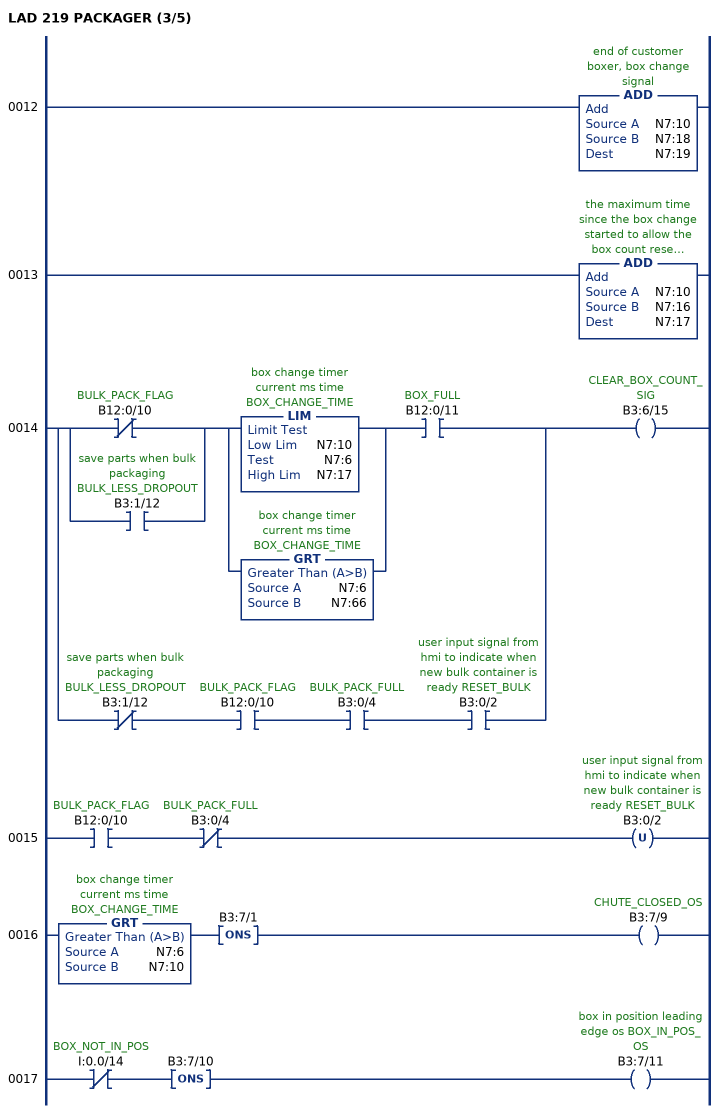
% Rung: 12 %
SOR ADD N7:10 N7:18 N7:19 EOR
%   N7:10  CHUTE_CLOSED_TIME  "time at which chute door is considered closed" %
%   N7:18  CHANGE_BOX_SIG_TIME  "customer boxer change box signal time" %
%   N7:19  "end of customer boxer, box change signal" %
% Rung: 13 %
SOR ADD N7:10 N7:16 N7:17 EOR
%   N7:10  CHUTE_CLOSED_TIME  "time at which chute door is considered closed" %
%   N7:16  RESET_COUNT_SIG_TIME  "maximum length of time to hold box count reset signal on" %
%   N7:17  "the maximum time since the box change started to allow the box count reset signal" %
% Rung: 14 %
SOR BST BST XIO B12:0/10 NXB XIC B3:1/12 BND BST LIM N7:10 N7:6 N7:17 NXB GRT N7:6 N7:66 BND XIC B12:0/11 NXB XIO B3:1/12 XIC B12:0/10 XIC B3:0/4 XIC B3:0/2 BND OTE B3:6/15 EOR
%   B12:0/10  BULK_PACK_FLAG %
%   B3:1/12  BULK_LESS_DROPOUT  "save parts when bulk packaging" %
%   N7:10  CHUTE_CLOSED_TIME  "time at which chute door is considered closed" %
%   N7:6  BOX_CHANGE_TIME  "box change timer current ms time" %
%   N7:17  "the maximum time since the box change started to allow the box count reset signal" %
%   B12:0/11  BOX_FULL %
%   B3:0/4  BULK_PACK_FULL %
%   B3:0/2  RESET_BULK  "user input signal from hmi to indicate when new bulk container is ready" %
%   B3:6/15  CLEAR_BOX_COUNT_SIG %
% Rung: 15 %
SOR XIC B12:0/10 XIO B3:0/4 OTU B3:0/2 EOR
%   B12:0/10  BULK_PACK_FLAG %
%   B3:0/4  BULK_PACK_FULL %
%   B3:0/2  RESET_BULK  "user input signal from hmi to indicate when new bulk container is ready" %
% Rung: 16 %
SOR GRT N7:6 N7:10 ONS B3:7/1 OTE B3:7/9 EOR
%   N7:6  BOX_CHANGE_TIME  "box change timer current ms time" %
%   N7:10  CHUTE_CLOSED_TIME  "time at which chute door is considered closed" %
%   B3:7/9  CHUTE_CLOSED_OS %
% Rung: 17 %
SOR XIO I:0.0/14 ONS B3:7/10 OTE B3:7/11 EOR
%   I:0.0/14  BOX_NOT_IN_POS %
%   B3:7/11  BOX_IN_POS_OS  "box in position leading edge os" %

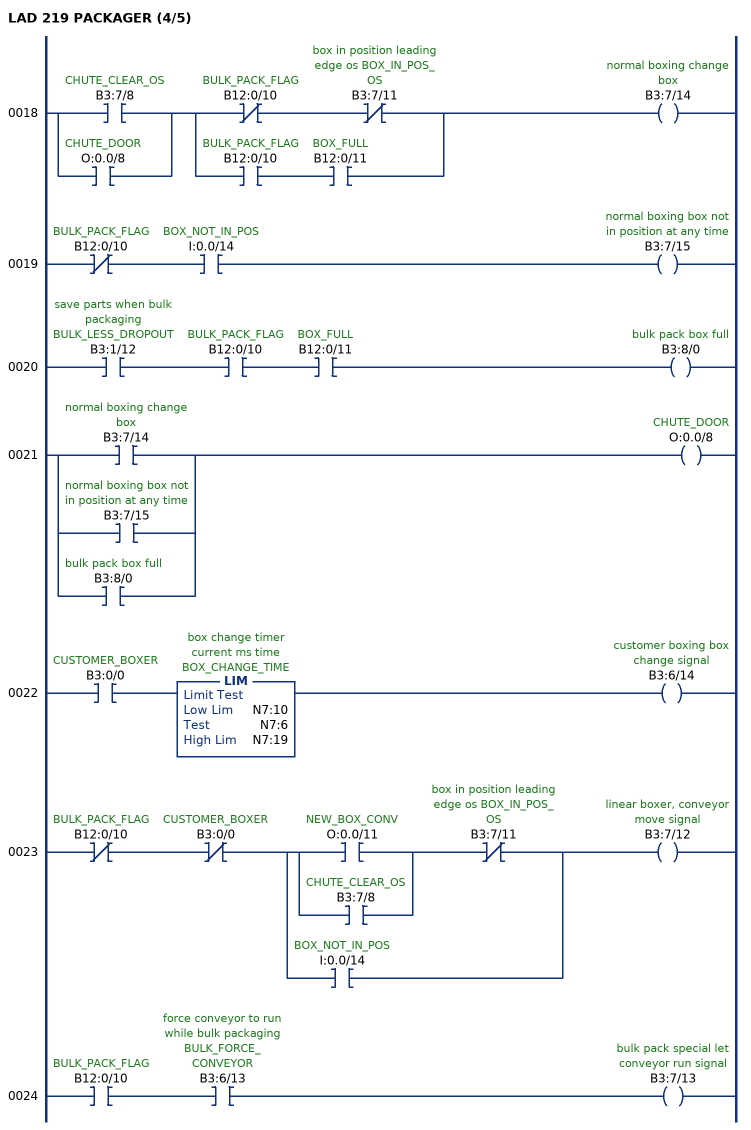
% Rung: 18 %
SOR BST XIC B3:7/8 NXB XIC O:0.0/8 BND BST XIO B12:0/10 XIO B3:7/11 NXB XIC B12:0/10 XIC B12:0/11 BND OTE B3:7/14 EOR
%   B3:7/8  CHUTE_CLEAR_OS %
%   O:0.0/8  CHUTE_DOOR %
%   B12:0/10  BULK_PACK_FLAG %
%   B3:7/11  BOX_IN_POS_OS  "box in position leading edge os" %
%   B12:0/11  BOX_FULL %
%   B3:7/14  "normal boxing change box" %
% Rung: 19 %
SOR XIO B12:0/10 XIC I:0.0/14 OTE B3:7/15 EOR
%   B12:0/10  BULK_PACK_FLAG %
%   I:0.0/14  BOX_NOT_IN_POS %
%   B3:7/15  "normal boxing box not in position at any time" %
% Rung: 20 %
SOR XIC B3:1/12 XIC B12:0/10 XIC B12:0/11 OTE B3:8/0 EOR
%   B3:1/12  BULK_LESS_DROPOUT  "save parts when bulk packaging" %
%   B12:0/10  BULK_PACK_FLAG %
%   B12:0/11  BOX_FULL %
%   B3:8/0  "bulk pack box full" %
% Rung: 21 %
SOR BST XIC B3:7/14 NXB XIC B3:7/15 NXB XIC B3:8/0 BND OTE O:0.0/8 EOR
%   B3:7/14  "normal boxing change box" %
%   B3:7/15  "normal boxing box not in position at any time" %
%   B3:8/0  "bulk pack box full" %
%   O:0.0/8  CHUTE_DOOR %
% Rung: 22 %
SOR XIC B3:0/0 LIM N7:10 N7:6 N7:19 OTE B3:6/14 EOR
%   B3:0/0  CUSTOMER_BOXER %
%   N7:10  CHUTE_CLOSED_TIME  "time at which chute door is considered closed" %
%   N7:6  BOX_CHANGE_TIME  "box change timer current ms time" %
%   N7:19  "end of customer boxer, box change signal" %
%   B3:6/14  "customer boxing box change signal" %
% Rung: 23 %
SOR XIO B12:0/10 XIO B3:0/0 BST BST XIC O:0.0/11 NXB XIC B3:7/8 BND XIO B3:7/11 NXB XIC I:0.0/14 BND OTE B3:7/12 EOR
%   B12:0/10  BULK_PACK_FLAG %
%   B3:0/0  CUSTOMER_BOXER %
%   O:0.0/11  NEW_BOX_CONV %
%   B3:7/8  CHUTE_CLEAR_OS %
%   B3:7/11  BOX_IN_POS_OS  "box in position leading edge os" %
%   I:0.0/14  BOX_NOT_IN_POS %
%   B3:7/12  "linear boxer, conveyor move signal" %
% Rung: 24 %
SOR XIC B12:0/10 XIC B3:6/13 OTE B3:7/13 EOR
%   B12:0/10  BULK_PACK_FLAG %
%   B3:6/13  BULK_FORCE_CONVEYOR  "force conveyor to run while bulk packaging" %
%   B3:7/13  "bulk pack special let conveyor run signal" %

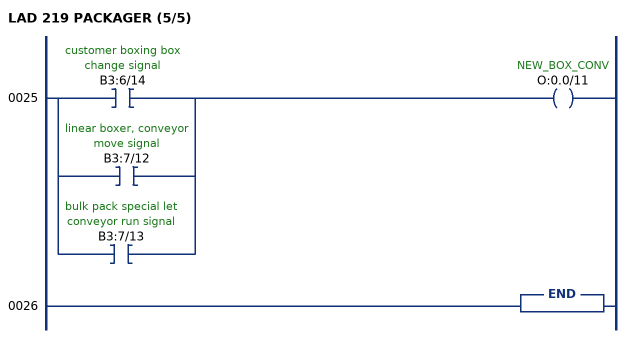
% Rung: 25 %
SOR BST XIC B3:6/14 NXB XIC B3:7/12 NXB XIC B3:7/13 BND OTE O:0.0/11 EOR
%   B3:6/14  "customer boxing box change signal" %
%   B3:7/12  "linear boxer, conveyor move signal" %
%   B3:7/13  "bulk pack special let conveyor run signal" %
%   O:0.0/11  NEW_BOX_CONV %
% Rung: 26 %
SOR END EOR

LADDER 220 "NO PACKAGE"
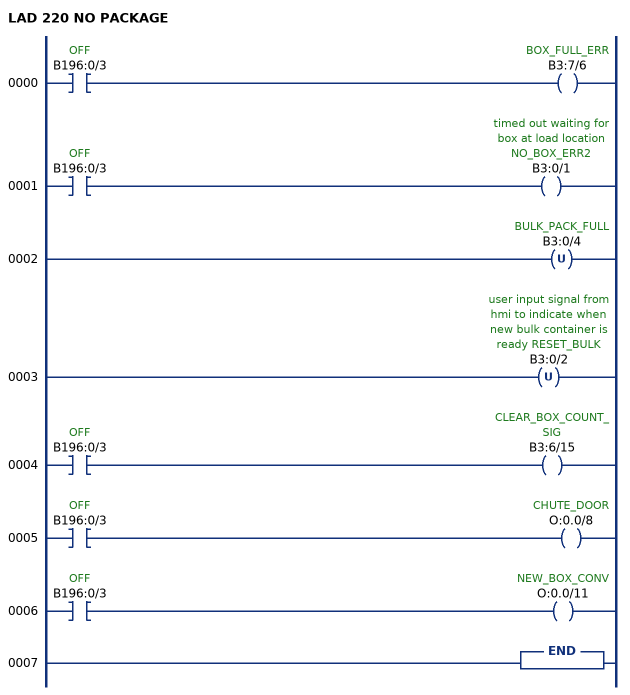
% Rung: 0 %
SOR XIC B196:0/3 OTE B3:7/6 EOR
%   B196:0/3  OFF %
%   B3:7/6  BOX_FULL_ERR %
% Rung: 1 %
SOR XIC B196:0/3 OTE B3:0/1 EOR
%   B196:0/3  OFF %
%   B3:0/1  NO_BOX_ERR2  "timed out waiting for box at load location" %
% Rung: 2 %
SOR OTU B3:0/4 EOR
%   B3:0/4  BULK_PACK_FULL %
% Rung: 3 %
SOR OTU B3:0/2 EOR
%   B3:0/2  RESET_BULK  "user input signal from hmi to indicate when new bulk container is ready" %
% Rung: 4 %
SOR XIC B196:0/3 OTE B3:6/15 EOR
%   B196:0/3  OFF %
%   B3:6/15  CLEAR_BOX_COUNT_SIG %
% Rung: 5 %
SOR XIC B196:0/3 OTE O:0.0/8 EOR
%   B196:0/3  OFF %
%   O:0.0/8  CHUTE_DOOR %
% Rung: 6 %
SOR XIC B196:0/3 OTE O:0.0/11 EOR
%   B196:0/3  OFF %
%   O:0.0/11  NEW_BOX_CONV %
% Rung: 7 %
SOR END EOR

LADDER 222 "RATE1"
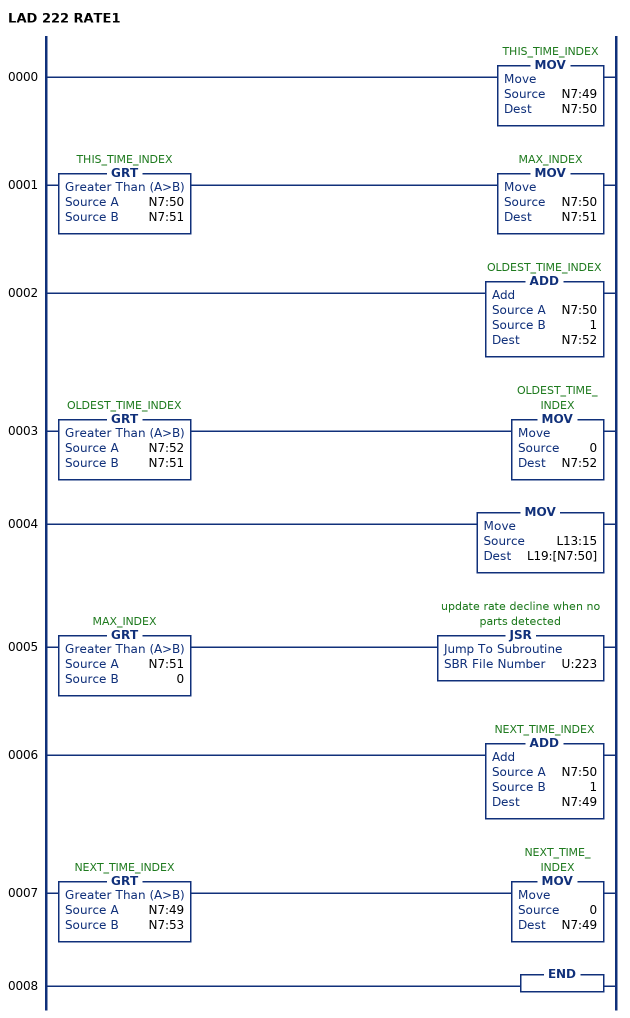
% Rung: 0 %
SOR MOV N7:49 N7:50 EOR
%   N7:49  NEXT_TIME_INDEX %
%   N7:50  THIS_TIME_INDEX %
% Rung: 1 %
SOR GRT N7:50 N7:51 MOV N7:50 N7:51 EOR
%   N7:50  THIS_TIME_INDEX %
%   N7:51  MAX_INDEX %
% Rung: 2 %
SOR ADD N7:50 1 N7:52 EOR
%   N7:50  THIS_TIME_INDEX %
%   N7:52  OLDEST_TIME_INDEX %
% Rung: 3 %
SOR GRT N7:52 N7:51 MOV 0 N7:52 EOR
%   N7:52  OLDEST_TIME_INDEX %
%   N7:51  MAX_INDEX %
% Rung: 4 %
SOR MOV L13:15 L19:[N7:50] EOR
%   L13:15  THE_TIME %
%   N7:50  THIS_TIME_INDEX %
% Rung: 5 %
SOR GRT N7:51 0 JSR U:223 EOR
%   N7:51  MAX_INDEX %
%   U:223  "update rate decline when no parts detected" %
% Rung: 6 %
SOR ADD N7:50 1 N7:49 EOR
%   N7:50  THIS_TIME_INDEX %
%   N7:49  NEXT_TIME_INDEX %
% Rung: 7 %
SOR GRT N7:49 N7:53 MOV 0 N7:49 EOR
%   N7:49  NEXT_TIME_INDEX %
%   N7:53  UPPER_INDEX_LIMIT %
% Rung: 8 %
SOR END EOR

LADDER 223 "RATE2"
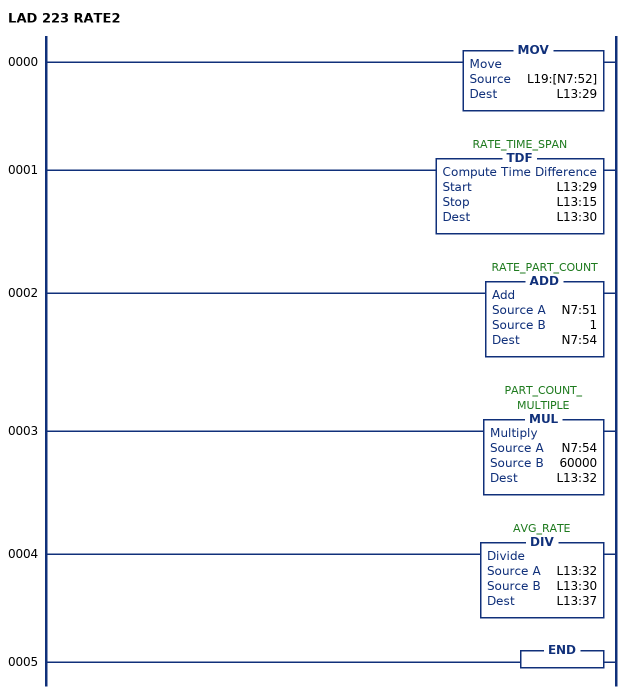
% Rung: 0 %
SOR MOV L19:[N7:52] L13:29 EOR
%   N7:52  OLDEST_TIME_INDEX %
% Rung: 1 %
SOR TDF L13:29 L13:15 L13:30 EOR
%   L13:15  THE_TIME %
%   L13:30  RATE_TIME_SPAN %
% Rung: 2 %
SOR ADD N7:51 1 N7:54 EOR
%   N7:51  MAX_INDEX %
%   N7:54  RATE_PART_COUNT %
% Rung: 3 %
SOR MUL N7:54 60000 L13:32 EOR
%   N7:54  RATE_PART_COUNT %
%   L13:32  PART_COUNT_MULTIPLE %
% Rung: 4 %
SOR DIV L13:32 L13:30 L13:37 EOR
%   L13:32  PART_COUNT_MULTIPLE %
%   L13:30  RATE_TIME_SPAN %
%   L13:37  AVG_RATE %
% Rung: 5 %
SOR END EOR

LADDER 224 "RESET RATE"
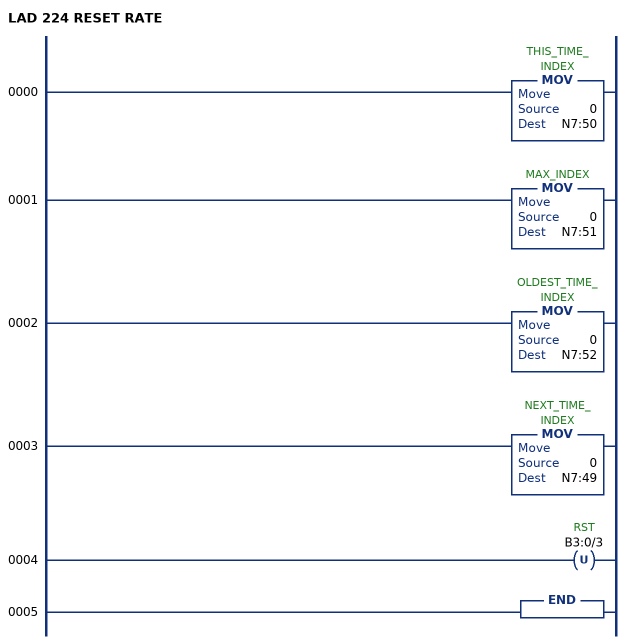
% Rung: 0 %
SOR MOV 0 N7:50 EOR
%   N7:50  THIS_TIME_INDEX %
% Rung: 1 %
SOR MOV 0 N7:51 EOR
%   N7:51  MAX_INDEX %
% Rung: 2 %
SOR MOV 0 N7:52 EOR
%   N7:52  OLDEST_TIME_INDEX %
% Rung: 3 %
SOR MOV 0 N7:49 EOR
%   N7:49  NEXT_TIME_INDEX %
% Rung: 4 %
SOR OTU B3:0/3 EOR
%   B3:0/3  RST %
% Rung: 5 %
SOR END EOR

LADDER 240 "NP STOP"
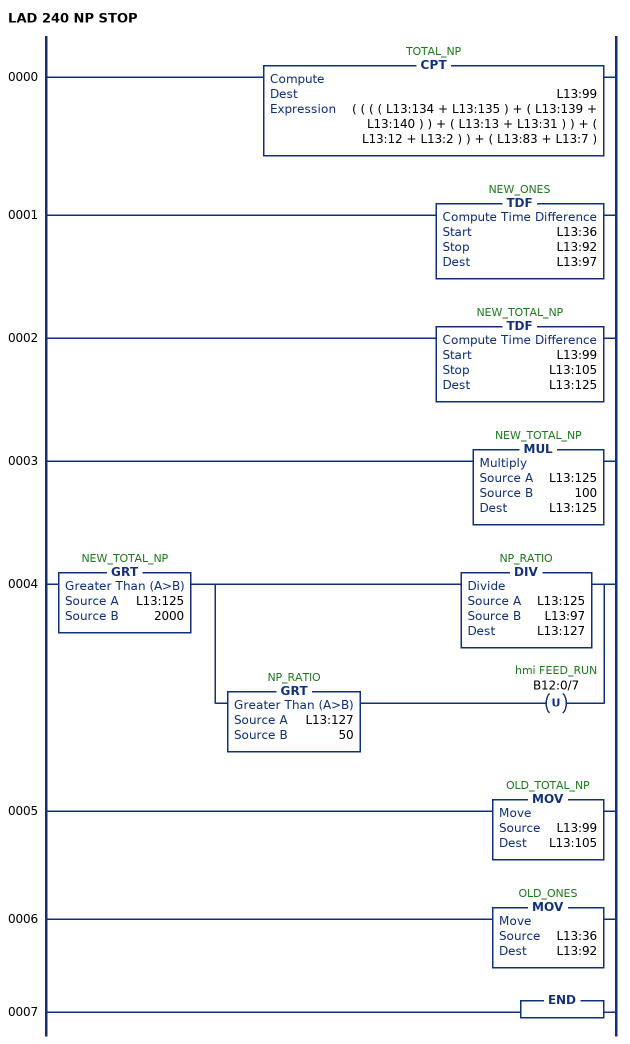
% Rung: 0 %
SOR CPT L13:99 " ( ( ( ( L13:134 + L13:135 ) + ( L13:139 + L13:140 ) ) + ( L13:13 + L13:31 ) ) + ( L13:12 + L13:2 ) ) + ( L13:83 + L13:7 ) " EOR
%   L13:99  TOTAL_NP %
%   L13:134  "too wide bottom" %
%   L13:135  "too close bottom" %
%   L13:139  "too close top count" %
%   L13:140  "too wide top count" %
%   L13:13  SKIP1  "skipped 1 count" %
%   L13:31  SKIP5  "skipped 5 count" %
%   L13:12  SKIP6  "skipped 6 count" %
%   L13:2  INS1_FAIL_COUNT %
%   L13:83  INS5_FAIL_COUNT %
%   L13:7  INS6_FAIL_COUNT %
% Rung: 1 %
SOR TDF L13:36 L13:92 L13:97 EOR
%   L13:36  ONES %
%   L13:92  OLD_ONES %
%   L13:97  NEW_ONES %
% Rung: 2 %
SOR TDF L13:99 L13:105 L13:125 EOR
%   L13:99  TOTAL_NP %
%   L13:105  OLD_TOTAL_NP %
%   L13:125  NEW_TOTAL_NP %
% Rung: 3 %
SOR MUL L13:125 100 L13:125 EOR
%   L13:125  NEW_TOTAL_NP %
% Rung: 4 %
SOR GRT L13:125 2000 BST DIV L13:125 L13:97 L13:127 NXB GRT L13:127 50 OTU B12:0/7 BND EOR
%   L13:125  NEW_TOTAL_NP %
%   L13:97  NEW_ONES %
%   L13:127  NP_RATIO %
%   B12:0/7  FEED_RUN  "hmi" %
% Rung: 5 %
SOR MOV L13:99 L13:105 EOR
%   L13:99  TOTAL_NP %
%   L13:105  OLD_TOTAL_NP %
% Rung: 6 %
SOR MOV L13:36 L13:92 EOR
%   L13:36  ONES %
%   L13:92  OLD_ONES %
% Rung: 7 %
SOR END EOR

LADDER 246 "SPEED BOT"    % high speed %
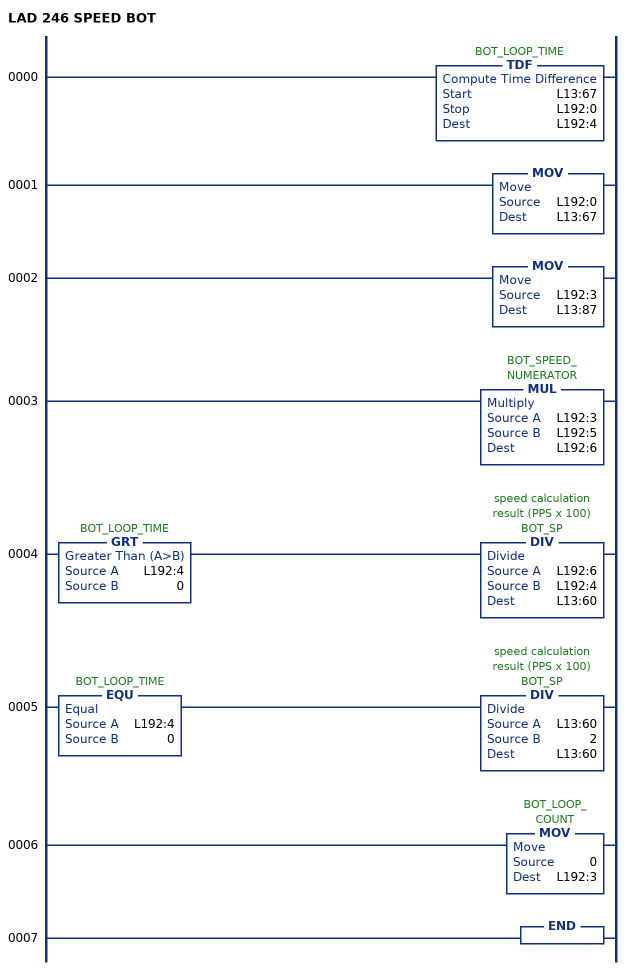
% Rung: 0 %
SOR TDF L13:67 L192:0 L192:4 EOR
%   L192:0  BOT_THIS_TIME  "rtc bot belt movement event time" %
%   L192:4  BOT_LOOP_TIME %
% Rung: 1 %
SOR MOV L192:0 L13:67 EOR
%   L192:0  BOT_THIS_TIME  "rtc bot belt movement event time" %
% Rung: 2 %
SOR MOV L192:3 L13:87 EOR
%   L192:3  BOT_LOOP_COUNT %
% Rung: 3 %
SOR MUL L192:3 L192:5 L192:6 EOR
%   L192:3  BOT_LOOP_COUNT %
%   L192:5  TKS_PER_SECOND %
%   L192:6  BOT_SPEED_NUMERATOR %
% Rung: 4 %
SOR GRT L192:4 0 DIV L192:6 L192:4 L13:60 EOR
%   L192:4  BOT_LOOP_TIME %
%   L192:6  BOT_SPEED_NUMERATOR %
%   L13:60  BOT_SP  "speed calculation result (PPS x 100)" %
% Rung: 5 %
SOR EQU L192:4 0 DIV L13:60 2 L13:60 EOR
%   L192:4  BOT_LOOP_TIME %
%   L13:60  BOT_SP  "speed calculation result (PPS x 100)" %
% Rung: 6 %
SOR MOV 0 L192:3 EOR
%   L192:3  BOT_LOOP_COUNT %
% Rung: 7 %
SOR END EOR

LADDER 248 "SPEED TOP"    % high speed %
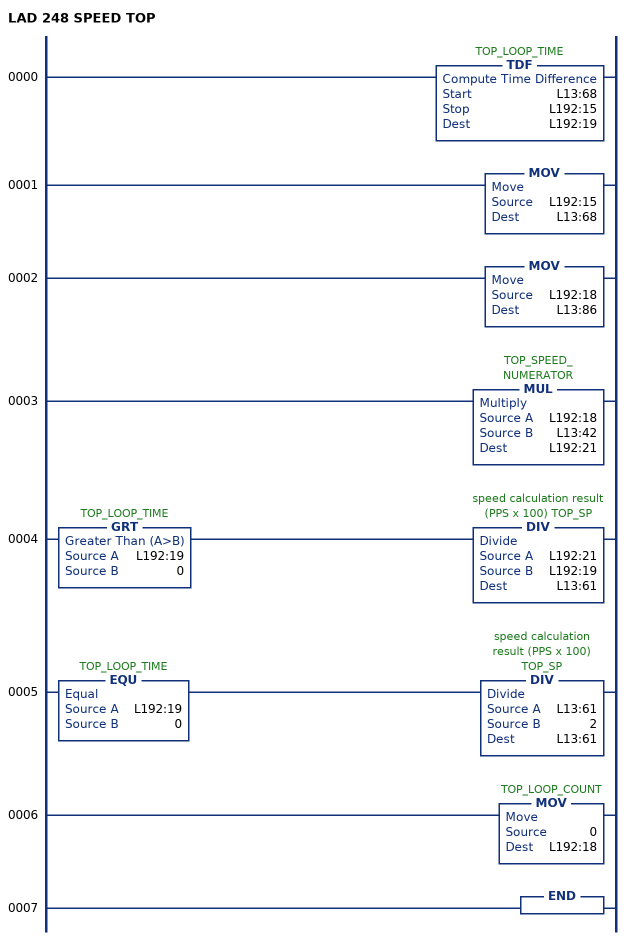
% Rung: 0 %
SOR TDF L13:68 L192:15 L192:19 EOR
%   L192:15  TOP_THIS_TIME  "rtc top belt movement event time" %
%   L192:19  TOP_LOOP_TIME %
% Rung: 1 %
SOR MOV L192:15 L13:68 EOR
%   L192:15  TOP_THIS_TIME  "rtc top belt movement event time" %
% Rung: 2 %
SOR MOV L192:18 L13:86 EOR
%   L192:18  TOP_LOOP_COUNT %
% Rung: 3 %
SOR MUL L192:18 L13:42 L192:21 EOR
%   L192:18  TOP_LOOP_COUNT %
%   L192:21  TOP_SPEED_NUMERATOR %
% Rung: 4 %
SOR GRT L192:19 0 DIV L192:21 L192:19 L13:61 EOR
%   L192:19  TOP_LOOP_TIME %
%   L192:21  TOP_SPEED_NUMERATOR %
%   L13:61  TOP_SP  "speed calculation result (PPS x 100)" %
% Rung: 5 %
SOR EQU L192:19 0 DIV L13:61 2 L13:61 EOR
%   L192:19  TOP_LOOP_TIME %
%   L13:61  TOP_SP  "speed calculation result (PPS x 100)" %
% Rung: 6 %
SOR MOV 0 L192:18 EOR
%   L192:18  TOP_LOOP_COUNT %
% Rung: 7 %
SOR END EOR

LADDER 250 "P BOT"    % high speed %
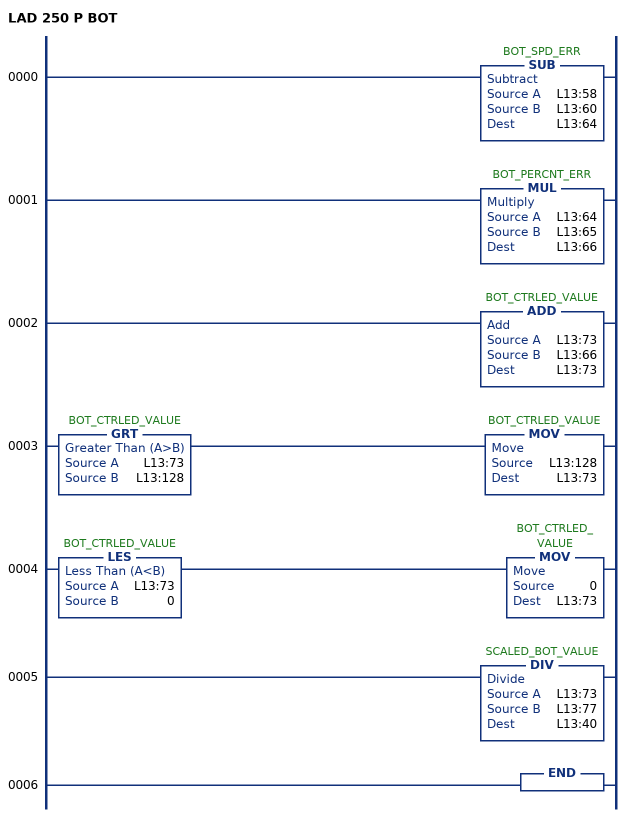
% Rung: 0 %
SOR SUB L13:58 L13:60 L13:64 EOR
%   L13:58  BOT_SPD_SETPOINT %
%   L13:60  BOT_SP  "speed calculation result (PPS x 100)" %
%   L13:64  BOT_SPD_ERR %
% Rung: 1 %
SOR MUL L13:64 L13:65 L13:66 EOR
%   L13:64  BOT_SPD_ERR %
%   L13:65  POS5SHIFT %
%   L13:66  BOT_PERCNT_ERR %
% Rung: 2 %
SOR ADD L13:73 L13:66 L13:73 EOR
%   L13:73  BOT_CTRLED_VALUE %
%   L13:66  BOT_PERCNT_ERR %
% Rung: 3 %
SOR GRT L13:73 L13:128 MOV L13:128 L13:73 EOR
%   L13:73  BOT_CTRLED_VALUE %
%   L13:128  "how much top has shifted since measurment" %
% Rung: 4 %
SOR LES L13:73 0 MOV 0 L13:73 EOR
%   L13:73  BOT_CTRLED_VALUE %
% Rung: 5 %
SOR DIV L13:73 L13:77 L13:40 EOR
%   L13:73  BOT_CTRLED_VALUE %
%   L13:40  SCALED_BOT_VALUE %
% Rung: 6 %
SOR END EOR

LADDER 252 "P TOP"    % high speed %
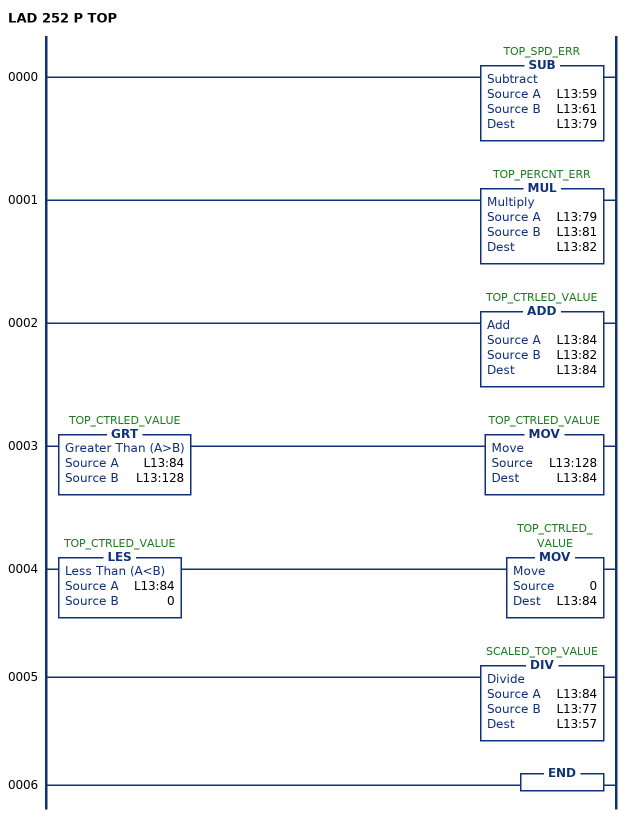
% Rung: 0 %
SOR SUB L13:59 L13:61 L13:79 EOR
%   L13:59  TOP_SPD_SETPOINT %
%   L13:61  TOP_SP  "speed calculation result (PPS x 100)" %
%   L13:79  TOP_SPD_ERR %
% Rung: 1 %
SOR MUL L13:79 L13:81 L13:82 EOR
%   L13:79  TOP_SPD_ERR %
%   L13:81  TOP_FDBK_RATIO %
%   L13:82  TOP_PERCNT_ERR %
% Rung: 2 %
SOR ADD L13:84 L13:82 L13:84 EOR
%   L13:84  TOP_CTRLED_VALUE %
%   L13:82  TOP_PERCNT_ERR %
% Rung: 3 %
SOR GRT L13:84 L13:128 MOV L13:128 L13:84 EOR
%   L13:84  TOP_CTRLED_VALUE %
%   L13:128  "how much top has shifted since measurment" %
% Rung: 4 %
SOR LES L13:84 0 MOV 0 L13:84 EOR
%   L13:84  TOP_CTRLED_VALUE %
% Rung: 5 %
SOR DIV L13:84 L13:77 L13:57 EOR
%   L13:84  TOP_CTRLED_VALUE %
%   L13:57  SCALED_TOP_VALUE %
% Rung: 6 %
SOR END EOR

LADDER 254 "TOTALCOUNT"
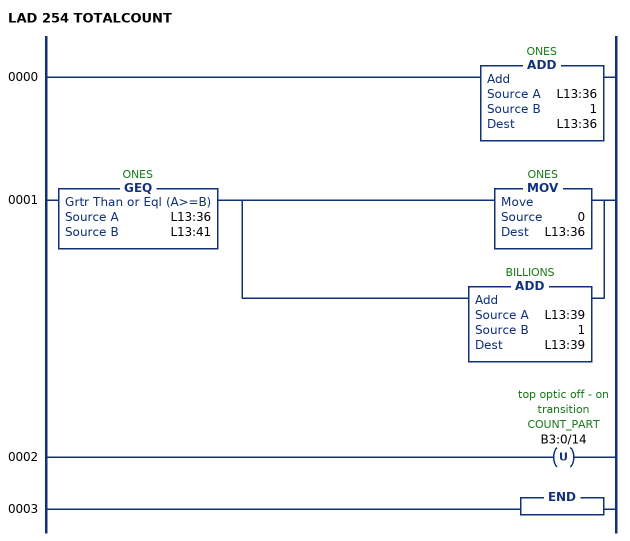
% Rung: 0 %
SOR ADD L13:36 1 L13:36 EOR
%   L13:36  ONES %
% Rung: 1 %
SOR GEQ L13:36 L13:41 BST MOV 0 L13:36 NXB ADD L13:39 1 L13:39 BND EOR
%   L13:36  ONES %
%   L13:41  "skipped count change in the last 3 seconds" %
%   L13:39  BILLIONS %
% Rung: 2 %
SOR OTU B3:0/14 EOR
%   B3:0/14  COUNT_PART  "top optic off - on transition" %
% Rung: 3 %
SOR END EOR

OTHER DOCUMENTED ADDRESSES
  I:0.0/0  TOPENC
  I:0.0/4  BOTENC
  I:0.1/1  "spare"
  PFILE:6  "check for part jams"
  PFILE:10  "Bottom belt HSC"
  PFILE:12  "Top belt HSC"
  Q2:55  END_OF_MAIN

COMMENTS NOT ATTACHED TO A CURRENT RUNG
  N17:8: ****************************************************************************************************************
    I can not find anywhere in the program where the "Test Spacing From Pickup to Trigger is activated indicating to me that this entire function must not be doing anything in this program at this time.
    ****************************************************************************************************************
  T20:2: The timer used to verify that the part that triggered the top laser optic has passed the bottom camer. needs to be count
  T20:2.ACC: This rung is starting a timer that should be activated directly before the laser optic part presense sensor on the top conveyer and should cause the top optic to be ignored if the bottom camera system didn't pass. however other arrangements must be made if the bottom camera isn't going to be used as is the case with a nut inspection.
  B22:0/0: ***********************
     Bottom Part Syncronizing Logic
    ***********************
    
    This is the point at the bottom of the top conveyor where the part jumps from the bottom conveyor.  This system will then track the part through the top system to the point of the laser optic in order to verify that the part in question has passed the bottom inspection.  I believe that we NEED to include FAILING inspections to eliminate the possibility of a out of position part from passing. LW 072010
  C5:4: tempory counting to verify pass part count with boxing part count.
  N7:25: 1050
  B23:0/0: Yet another bit shift load with data in the part position indicating that there was a bottom system part pass as well as a top system part present at this location.
    
    verified works w/bypassed 071910 and unbypassed 072010
  I:0.0/8: special rung for testing. This rung can simulate a pass signal. It will not be timed correctly.
  F8:13: *************************
    Loads Side Camera Passing data into a bit shift
    *************************
    
    loads passing data bit into passing data bit shift register at the part present cl.
  B11:0/0: load part present bit shit with one shot data from the part present sensor
  N7:45: not fully functional because of part overlap but measurems the camera responce time when part inspections are not overlaping
  B3:6/1: ***********************
    Part Width and  Location
    ***********************
    
    Calculates the position of parts on the top belt by measureing the part width by calculating the number of belt movement pulses that occure when the optic is blocked and then devides that in half and add that to the optic location in the part presnet bit shift when the top optic is cleared.
  B9:0/[N7:47]: Remove any part present signals outside of expected location
  B9:0/[N7:50]: Remove any part present signals outside of expected location
  F19:0: Counter inside of a high speed counter interrupt counts the number of Bit Shifts that need to be processed in order to move the logic with the parts on the conveyor.
  F8:14: **************
    Bottom Top Camera Trigger
    *************
    
    Trigger Bottom Top Camera
  N10:4: test if boxing is connected
  T4:28: Check for buffer reset
  B3:11/3: After initial delay allow blow two start functioning
  RUNG000150-000041: transfer tracked part positon from trigger/acquire to the acquire/result
    capture acquire time
    reset process time
  RUNG000150-000039: Grab trigger/acquire position
    Grab acquire time
  RUNG000150-000038: acquire code
  RUNG000150-000035: fail count
  RUNG000150-000032: pass count
  RUNG000150-000025: pass code / Set pass bit in Bit Shift
    captures result position and processing time
    Unlatch pass bit
  RUNG000150-000018: pass, fail and acquire inputs
  RUNG000150-000016: wiped count
  RUNG000150-000014: clear data for time
  RUNG000150-000013: clear data for aquire time expired
  RUNG000150-000012: wipe stored part data if acq time expires
  RUNG000150-000011: trigger count
  L14:5: on when ok to run, rear off turns both off
  L14:2: off when ok to run
  L14:3: off when ok to run
  L14:8: on when ok for run
  L13:165: maximum q i1
  N7:76: removed relieance on trigger signal
  N197:20/0: Passes deformed head blowoff command to TOP PLC where solenoid output is located.
  L13:163: maximum average q
  L13:162: maximum q
  N7:47: ***********************************************************************************************************************************************************
    From side
    ***********************************************************************************************************************************************************
    
    removed relieance on trigger signal
  B3:10/1: prevents momentary signals from box present sensor from tripping the logic for box not present
    
    This is in responce to a problem created by the sensor occasionally turning on as if no box was in its path when there is a box present.
  B3:6/2: IF PROCESSING FAULT OCURES AT COUNTER SENSOR; CLEAR THE BELT OF PASSING DATA
  L14:36: ****************  nEEDS fIXING  **********************
  L14:23: ****************  nEEDS fIXING  **********************
  RUNG000010-000018: Remove any part present signals outside of expected location
  RUNG000010-000014: ****
                      Zeros out the non passing part count when one passes
    ****
  T4:26: Check for buffer reset
  T4:27: Check for buffer reset
  RUNG000125-000011: trigger count
  RUNG000125-000012: wipe stored part data if acq time expires
  RUNG000125-000013: clear data for aquire time expired
  RUNG000125-000014: clear data for time
  RUNG000125-000016: wiped count
  RUNG000125-000018: pass, fail and acquire inputs
  RUNG000125-000025: pass code / Set pass bit in Bit Shift
    captures result position and processing time
    Unlatch pass bit
  RUNG000125-000026: Grab trigger/acquire position
    Grab acquire time
  RUNG000125-000027: transfer tracked part positon from trigger/acquire to the acquire/result
    capture acquire time
    reset process time
  RUNG000125-000029: Set pass bit in Bit Shift
    captures result position and processing time
    Unlatch pass bit

REVISION NOTES
  13: updated count reset
  14: added io moduals
  15: multiple steps toward new hmi integration
  21: test

DATA TABLE (non-zero values as saved)
DATA B3
% B3:0 % 0XA0A0 0X0040 0X4005 0XA000 0XDE7D 0X1540 0X0183 0X0420 0X4924 0X0000
% B3:10 % 0X2041 0X0846 0X2000 0X0000
DATA T4
% .PRE .ACC %
% T4:0 % 0 1
% T4:1 % 150 0
% T4:2 % 400 0
% T4:3 % 333 257
% T4:4 % 300 300
% T4:5 % 250 0
% T4:6 % 10 10
% T4:7 % 666 0
% T4:8 % 20 7
% T4:9 % 50 21
% T4:10 % 200 200
% T4:11 % 111 0
% T4:12 % 20 20
% T4:13 % 250 0
% T4:14 % 666 0
% T4:15 % 1000 1000
% T4:16 % 11 0
% T4:17 % 100 35
% T4:18 % 15 15
% T4:19 % 300 0
% T4:20 % 200 0
% T4:21 % 200 0
% T4:22 % 200 0
% T4:23 % 250 0
% T4:24 % 666 0
% T4:25 % 50 0
% T4:26 % 250 0
% T4:27 % 250 0
% T4:28 % 250 0
% T4:29 % 5000 0
% T4:30 % 333 251
% T4:31 % 333 217
% T4:32 % 69 0
DATA C5
% .PRE .ACC %
% C5:0 % 32766 0
DATA R6
% .LEN .POS %
% R6:0 % 1250 0
% R6:1 % 1250 0
% R6:2 % 1024 0
% R6:3 % 1024 0
% R6:4 % 1250 0
% R6:5 % 1250 0
% R6:6 % 1250 0
% R6:7 % 1024 0
% R6:8 % 1024 0
% R6:9 % 3 0
% R6:10 % 2000 0
% R6:11 % 1024 0
% R6:12 % 10 0
% R6:13 % 10 0
% R6:14 % 10 0
% R6:15 % 10 0
% R6:16 % 1250 0
% R6:17 % 2000 0
% R6:18 % 1024 0
% R6:19 % 10 0
DATA N7
% N7:0 % 32767 5 950 300 300 400 0 120 500 500
% N7:10 % 1000 55 0 2 20 20 1000 2000 50 1050
% N7:20 % 32767 333 10 333 333 46 32 0 32 250
% N7:30 % 666 32767 150 0 0 1321 83 21 0 21
% N7:40 % 0 30 0 30 1337 1520 1343 1555 434 6
% N7:50 % 5 16 6 16 17 0 0 0 32766 0
% N7:60 % 1250 2000 1024 946 1034 1024 4999 15 400 0
% N7:70 % 0 0 23 27738 32767 0 122 0 16 0
% N7:80 % 0 6 95 0 0 0 5 500 0 0
% N7:90 % 2011 4 4 12 1 0 0 0 0 1600
% N7:100 % 1003 90 110 100 175 25 0 0 0 0
DATA F8
% F8:0 % 6 1 23807 499 0.23807
% F8:5 % 0 0 500 1.9 2
% F8:10 % 1 0.08897486 3058 101 63.26563
% F8:15 % 37.73437 4040 2 0 0
% F8:20 % 0 0.02 0 1 0
% F8:25 % 0 932781 0.222 279.6551 848597
% F8:30 % 0 170 0.03 38 852060
% F8:35 % 0 0 0 0 77
% F8:40 % 101 37.73437 0 100 1
% F8:45 % 1 2 0.21455 0 0
% F8:50 % 0 0 1 0 1
% F8:55 % 2000000 -221 0 0 0
% F8:95 % 0 0 0 492 4.92
DATA B12
% B12:0 % 0X0155 0X0000 0X0000 0X0000 0X0000 0X0000 0X0000 0X0000 0X0000 0X0000
DATA L13
% L13:0 % 0 0 0 5 -543897413
% L13:5 % 1257 0 50 355917 337
% L13:10 % 1330117815 65 4966 198 30
% L13:15 % -543541496 -2147483648 2147483647 2147483647 82058
% L13:20 % 1330117815 1335454288 777 1330117815 100
% L13:25 % 500 30 1 -4 -545975105
% L13:30 % 2432869 1640 1020000 -545724706 444
% L13:35 % 62432 66524 0 0 0
% L13:40 % 0 1000000000 1000000 -545724734 0
% L13:45 % 60 300 0 28 1335333375
% L13:50 % 0 2183279 -545724712 0 60
% L13:55 % 0 2183257 344 0 500
% L13:60 % 0 504 28 600 0
% L13:65 % 100 0 12433395 131927108 -543897383
% L13:70 % 1335333385 26 10 0 1335333375
% L13:75 % 17 0 1000 -545724686 -4
% L13:80 % 26 74 -296 8 344176
% L13:85 % 121290 25 0 26483 1000
% L13:90 % 26616 0 66524 1000 0
% L13:95 % 60 144 0 25989 6862
% L13:100 % 1000 7 400 3 144
% L13:105 % 6862 4 1330104258 69 1330104248
% L13:110 % 10 30 10 1335333005 1335332993
% L13:115 % 1335333001 8 4 1335332997 53659
% L13:120 % 13 64 10 29 55298
% L13:125 % 0 1335333385 2147483647 3276500 121287
% L13:130 % 2 2 0 6 0
% L13:135 % 0 1000 121287 5 0
% L13:140 % 0 5 36 50 50
% L13:145 % 5 5 5 5 40
% L13:150 % 12 20 4 -4 65
% L13:155 % 0 -8 40 0 4589052
% L13:160 % 3 7 4 395082 53203921
% L13:165 % 3 189116 95 13 8150
% L13:170 % 55946610 30 72 54 0
% L13:175 % 0 0 42 23 38
% L13:180 % 176247033 25 99000 52866 644409
% L13:185 % 64 916459 92 627156 63
% L13:190 % 4 5 0 0 0
DATA F14
% F14:0 % 1.32889e-38 5747.126 1550 1550 1638.3
% F14:5 % 1638.3 1638.3 1638.3 0 0
DATA N15
% N15:0 % 6 846 1645 1330 1320 120 100 1178 942 10
% N15:10 % 58 717 0 0 0 0 1178 0 0 0
DATA L16
% L16:0 % 8 20 11 0 20
% L16:5 % 250 5000 5000 182 19
% L16:10 % 1256 18 2045 6599584 98
% L16:15 % 99 0 0 0 0
DATA L19
% L19:0 % -545726081 -545725988 -545725904 -545725812 -545725699
% L19:5 % -545725548 -545975105 -545975014 -545974931 -545974854
% L19:10 % -545974765 -545974662 -545974589 -545974492 -545726335
% L19:15 % -545726238 -545726161 0 0 0
DATA L28
% L28:0 % -544766662 -544766326 -544765991 -544765655 -544765319
% L28:5 % -544764983 -544764646 -544764309 -544763972 -544763637
% L28:10 % -544763301 -544762965 -544762629 -544762292 -544761956
% L28:15 % -544761621 -544761285 -544760950 -544760614 -544760278
% L28:20 % -544759941 -544759605 -544759269 -544758932 -544758595
% L28:25 % -543899765 -543899430 -543899094 -543898758 -543898421
% L28:30 % -543898085 -543897750 -543897413 -544772373 -544772037
% L28:35 % -544771701 -544771365 -544771029 -544770692 -544770357
% L28:40 % -544770020 -544769683 -544769346 -544769011 -544768675
% L28:45 % -544768340 -544768004 -544767669 -544767333 -544766998
DATA L29
% L29:0 % 1330117814 1330117814 1330117814 1330117814 1330117814
% L29:5 % 1330117814 1330117814 1330117814 1330117814 1330117814
% L29:10 % 1330117814 1330117814 1330117814 1330117814 1330117814
% L29:15 % 1330117814 1330117814 1330117814 1330117814 1330117814
% L29:20 % 1330117814 1330117814 1330117814 1330117814 1330117814
% L29:25 % 1330117815 1330117815 1330117815 1330117815 1330117815
% L29:30 % 1330117815 1330117815 1330117815 1330117814 1330117814
% L29:35 % 1330117814 1330117814 1330117814 1330117814 1330117814
% L29:40 % 1330117814 1330117814 1330117814 1330117814 1330117814
% L29:45 % 1330117814 1330117814 1330117814 1330117814 1330117814
DATA L30
% L30:0 % -545974680 -545974594 -545974504 -545974424 -545974359
% L30:5 % -545974284 -545974200 -545974110 -545974033 -545973942
% L30:10 % -545973846 -545973768 -545973672 -545725511 -545725414
% L30:15 % -545725339 -545725257 -545725168 -545725080 -545724993
% L30:20 % -545724878 -545724734 -545976970 -545976889 -545976807
% L30:25 % -545976716 -545976621 -545976541 -545976460 -545976374
% L30:30 % -545976275 -545976209 -545976134 -545976050 -545975972
% L30:35 % -545975888 -545975799 -545975731 -545975660 -545975570
% L30:40 % -545975486 -545975402 -545975324 -545975236 -545975159
% L30:45 % -545975086 -545974996 -545974910 -545974844 -545974764
DATA L31
% L31:0 % 1335219985 1335220024 1335220065 1335220101 1335220131
% L31:5 % 1335220165 1335220203 1335220244 1335220279 1335220320
% L31:10 % 1335220364 1335220399 1335220443 1335333023 1335333067
% L31:15 % 1335333101 1335333138 1335333178 1335333218 1335333258
% L31:20 % 1335333310 1335333375 1335218949 1335218986 1335219023
% L31:25 % 1335219064 1335219107 1335219143 1335219180 1335219218
% L31:30 % 1335219263 1335219293 1335219327 1335219365 1335219400
% L31:35 % 1335219438 1335219478 1335219509 1335219541 1335219582
% L31:40 % 1335219620 1335219658 1335219693 1335219733 1335219768
% L31:45 % 1335219801 1335219842 1335219881 1335219911 1335219947
DATA L32
% L32:0 % -545975380 -545975302 -545975214 -545975136 -545975064
% L32:5 % -545974974 -545974888 -545974822 -545974742 -545974659
% L32:10 % -545974572 -545974481 -545974402 -545974337 -545974262
% L32:15 % -545974178 -545974088 -545974011 -545973920 -545973823
% L32:20 % -545973747 -545973650 -545725489 -545725392 -545725316
% L32:25 % -545725235 -545725146 -545725058 -545724970 -545724856
% L32:30 % -545724712 -545976948 -545976867 -545976785 -545976694
% L32:35 % -545976599 -545976519 -545976437 -545976352 -545976253
% L32:40 % -545976187 -545976112 -545976028 -545975950 -545975866
% L32:45 % -545975777 -545975708 -545975638 -545975548 -545975464
DATA L33
% L33:0 % 1335219668 1335219703 1335219743 1335219778 1335219811
% L33:5 % 1335219852 1335219891 1335219921 1335219957 1335219995
% L33:10 % 1335220034 1335220075 1335220111 1335220141 1335220175
% L33:15 % 1335220213 1335220254 1335220289 1335220330 1335220374
% L33:20 % 1335220409 1335220453 1335333033 1335333077 1335333111
% L33:25 % 1335333148 1335333188 1335333228 1335333268 1335333320
% L33:30 % 1335333385 1335218959 1335218996 1335219033 1335219074
% L33:35 % 1335219117 1335219153 1335219190 1335219228 1335219273
% L33:40 % 1335219303 1335219337 1335219375 1335219410 1335219448
% L33:45 % 1335219488 1335219519 1335219551 1335219592 1335219630
DATA B35
% B35:70 % 0X0000 0X0000 0X0000 0X0000 0X0000 0X0000 0X0000 0X0000 0X0000 0XFFFF
% B35:80 % 0XFFFF 0XFFFF 0XE11F 0XC880 0X01FF 0X0000 0X0000 0X0020 0X0000 0X0C00
% B35:90 % 0X0000 0X0100 0X0004 0X0000 0X0002 0X0000 0X0000 0X0000 0X0000 0X0000
DATA B38
% B38:50 % 0X0000 0X0000 0X0000 0X0000 0X0000 0X0000 0X0000 0X0000 0X6000 0X01FF
% B38:60 % 0X0000 0X0000 0X0000 0X8800 0X0003 0X0000 0X0FFF 0X0000 0X0000 0X0000
% B38:120 % 0X0000 0X0000 0X0000 0X0000 0X0000 0X0000 0X0000 0X0002
DATA B40
% B40:50 % 0X0000 0X0000 0X0000 0X0000 0X0000 0X0000 0X0000 0X0000 0X6000 0X01FF
% B40:60 % 0X0000 0X0000 0X0000 0X8800 0X0003 0X0000 0X0FFF 0X0000 0X0000 0X0000
% B40:120 % 0X0000 0X0000 0X0000 0X0000 0X0000 0X0000 0X0000 0X0002
DATA L192
% L192:0 % 12433395 266932201 5055 0 0
% L192:5 % 1000000 0 999 999 8
% L192:10 % 0 0 0 78 17
% L192:15 % 132087500 332250347 860888 4 49456
% L192:20 % 180 25000000 0 0 0
DATA B196
% B196:0 % 0X0814 0X9FFE 0X0005 0X0000 0X0000 0X0000 0X0000 0X0000 0X0000 0X0000
% B196:30 % 0XE800 0X9BFF 0XEBFF 0XFFDF 0XFFFF 0X0000 0X0000 0X0000 0X0000 0X0000
DATA L199
% L199:0 % 1 0 0 0 0
